TEXTLIST TextList_Dialogs
  0 = 'Select the function'
  1 = 'Control Gears - Commands'
  2 = 'Control Gears - Addressing'
  3 = 'Control Gears - Parameters'
  4 = 'Control Gears - Groups'
  5 = 'Control Gears - Scenes'
  6 = 'Control Gears - Memory Pages'
  7 = 'Control Gears - Set Fading'
  8 = 'Control Gears - Device Type 1 (Emergency lighting)'
  9 = 'Control Gears - Device Type 4 (Incandescent lamp)'
  10 = 'Control Gears - Device Type 6 (LED)'
  11 = 'Control Gears - Device Type 7 (Switching)'
  12 = 'Control Devices - Addressing'
  13 = 'Control Devices - Parameters'
  15 = 'Control Devices - Device Type 1 (Push button)'
  16 = 'Control Devices - Device Type 2 (Absolute input)'
  17 = 'Control Devices - Device Type 3 (Occupancy sensor)'
  18 = 'Control Devices - Device Type 4 (Light sensor)'
  19 = 'Control Devices - Device Type 0 (Generic instance)'
  20 = 'Control Devices - Memory Pages'
  14 = 'Control Devices - Identify'
   = ''
END_TEXTLIST

(* stored: Version 1.1.0.1
   TextList TextList_Dialogs: Id {549a1fb5-0049-4732-ae1c-91ef7c52241f} *)
